TYPE Coordinate :
STRUCT
	X : LREAL;
	Y : LREAL;
END_STRUCT
END_TYPE

(* stored: Version 1.1.0.1
   DUT Coordinate: Id {f4188b48-0f81-459b-8804-da988f450db9} *)
